(* PLC project Unnamed, Unknown Unnamed 1 *)
(* stored: creationDateTime 2021-07-26T15:42:18, modificationDateTime 2021-08-02T14:58:00 *)

FUNCTION_BLOCK MoveArm
  VAR_INPUT
    ENABLE : BOOL := FALSE;
    SPEED : SINT := 0;
    TARGET : STRING := '0,0,0,0,0,0,0';
  END_VAR
  VAR_OUTPUT
    VALID : BOOL := FALSE;
    ERROR : BOOL := FALSE;
    ERRORCODE : SINT := 0;
  END_VAR
  VAR
    WAIT : SINT := 0;
  END_VAR

            {{
  int wait = GetFbVar(WAIT);
  bool enable = GetFbVar(ENABLE);
  int fd = open("/tmp/ArmControl.pipe",O_RDWR | O_NONBLOCK);
  if(wait==0 && enable){
    SetFbVar(WAIT, 1);
  }
  else if(wait == 1){
    char buf[200] = {"movePos;"};
    //SPEED
    int speed = GetFbVar(SPEED);
    strcat(buf, "1");
    //char *word = GetFbVar(TARGET).body;
    //sprintf(word, "%d", speed);
    //strcat(buf,word);
    strcat(buf,",");
    //Target
    char *word1 = GetFbVar(TARGET).body;
    strcat(buf,word1);
    strcat(buf,";");
    
    int ret = write(fd, buf, 200);
    if(ret > 0){
      SetFbVar(WAIT, 2);
    }
  }
  else if(wait == 2){
    char buf[200];
    int ret = read(fd, buf, 200);
    if(ret>0){
      if(buf[0]=='n'){
        //ERROR
        SetFbVar(ERROR, true);
        //1-digit error id
        SetFbVar(ERRORCODE, buf[1] - 48);
        SetFbVar(WAIT, 3);
      }
      else if(buf[0] == 'Y' && buf[2] == 'm' ){
        SetFbVar(VALID, true);
        SetFbVar(WAIT, 3);
      }
      else{
        write(fd, buf, 200);
      }
    }
  }
  else if((wait == 3) && !enable){
    
    SetFbVar(VALID, false);
    SetFbVar(ERROR, false);
    SetFbVar(ERRORCODE, 0);
    SetFbVar(WAIT, 0);
  }
  close(fd);
}}
          
END_FUNCTION_BLOCK

PROGRAM program0
  VAR
    SWITCH : BOOL;
    COUNTER : LINT := 0;
    ONE : LINT := 1;
    SPEED : SINT := 1;
    TARGET1 : STRING := '219.91,-332.00,289.34,0.21,0.66,-0.65,0.32';
    TARGET2 : STRING := '636.63,138.27,410.64,0.12,-0.72,0.07,-0.68';
    R_TRIG0 : R_TRIG;
    functionBlock1 : MoveArm;
    functionBlock0 : MoveArm;
    R_TRIG1 : R_TRIG;
  END_VAR
  VAR  (* added by the conversion: wires and edge detectors of the diagram *)
    _ADD11_ENO : BOOL;
    _ADD11_OUT : LINT;
  END_VAR

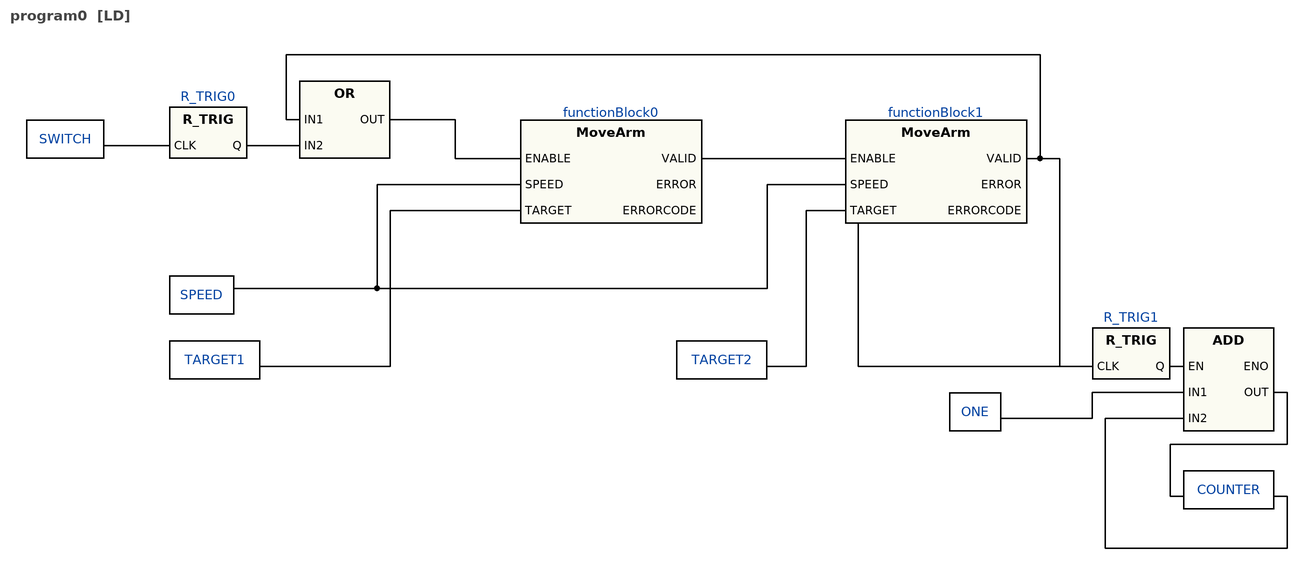
(* LD diagram, written out as Structured Text *)
functionBlock1(ENABLE := functionBlock0.VALID, SPEED := SPEED, TARGET := TARGET2);
R_TRIG0(CLK := SWITCH);
functionBlock0(ENABLE := functionBlock1.VALID OR R_TRIG0.Q, SPEED := SPEED, TARGET := TARGET1);
R_TRIG1(CLK := functionBlock0.VALID OR functionBlock1.VALID);
_ADD11_OUT := ADD(EN := R_TRIG1.Q, IN1 := ONE, IN2 := COUNTER, ENO => _ADD11_ENO);
IF _ADD11_ENO THEN COUNTER := _ADD11_OUT; END_IF;
END_PROGRAM

CONFIGURATION Config0
  RESOURCE Res0 ON PLC
    TASK task0(INTERVAL := T#20ms, PRIORITY := 0);
    PROGRAM instance0 WITH task0 : program0;
  END_RESOURCE
END_CONFIGURATION
